(* Logix 5000 project; controller Proyecto_APM vendor 1 type 14 code 156 rev 30.11; software revision 30.00 *)

TASK MainTask (continuous, watchdog 500 ms) : MainProgram

MODULES
   Local : vendor 1 type 14 code 156 (Compact 0, rev 30.11)
      Dis : 1769-IQ16 (Compact 4, rev 1.1, Input RPI 20 ms)
      DOs : vendor 1 type 7 code 86 (Compact 5, rev 2.1, Output RPI 20 ms)
END_MODULES

VAR_GLOBAL   (* controller tags *)
   BIn : BOOL := 1;
   BoFc1 : BOOL;
   BoIn : BOOL;
   BoPi : BOOL;
   BTr : BOOL;
   CaIn : BOOL;
   EmFc : BOOL;
   EmPi : BOOL;
   FFc1 : BOOL;
   FFc2 : BOOL;
   FFc3 : BOOL;
   FiFcI : BOOL;
   FiFcS : BOOL;
   FiPi : BOOL;
   HPi : BOOL;
   I : BOOL;
   PaPi1 : BOOL;
   PaPi2 : BOOL;
   PaPi3 : BOOL;
   PaTrI : BOOL;
   PaTrS : BOOL;
   PIn : BOOL;
   S : BOOL;
END_VAR

PROGRAM MainProgram   (* main routine MainRoutine *)
VAR
   BoFc2 : BOOL;
   BoFc3 : BOOL;
   CFc1 : BOOL;
   CFc2 : BOOL;
   CFc3 : BOOL;
   E0 : BOOL := 1;
   E11_0 : BOOL := 1;
   E11_1 : BOOL;
   E11_2 : BOOL;
   E11_3 : BOOL;
   E12_0 : BOOL := 1;
   E12_1 : BOOL;
   E12_2 : BOOL;
   E12_3 : BOOL;
   E13_0 : BOOL := 1;
   E13_1 : BOOL;
   E13_2 : BOOL;
   E13_3 : BOOL;
   E2_0 : BOOL := 1;
   E2_1 : BOOL;
   E2_2 : BOOL;
   E2_3 : BOOL;
   E31_0 : BOOL := 1;
   E31_1 : BOOL;
   E31_2 : BOOL;
   E31_3 : BOOL;
   E32_0 : BOOL := 1;
   E32_1 : BOOL;
   E32_2 : BOOL;
   E32_3 : BOOL;
   E33_0 : BOOL := 1;
   E33_1 : BOOL;
   E33_2 : BOOL;
   E33_3 : BOOL;
   E3_0 : BOOL;
   E3_1 : BOOL;
   E3_2 : BOOL;
   E4_0 : BOOL;
   E4_1 : BOOL := 1;
   E4_2 : BOOL;
   E4_3 : BOOL;
   E4_4 : BOOL;
   EmIn : BOOL;
   EmTr : BOOL;
   iBIn : BOOL := 1;
   iBoFc1 : BOOL;
   iBoFc2 : BOOL;
   iBoFc3 : BOOL;
   iBoIn : BOOL;
   iBoPi : BOOL;
   iBTr : BOOL;
   iCaIn : BOOL;
   iCFc1 : BOOL;
   iCFc2 : BOOL;
   iCFc3 : BOOL;
   iEmFc : BOOL;
   iEmIn : BOOL;
   iEmPi : BOOL;
   iEmTr : BOOL;
   iFFc1 : BOOL;
   iFFc2 : BOOL;
   iFFc3 : BOOL;
   iFiFcI : BOOL;
   iFiFcS : BOOL;
   iFiPi : BOOL;
   iHPi : BOOL;
   iPaPi1 : BOOL;
   iPaPi2 : BOOL;
   iPaPi3 : BOOL;
   iPaTrI : BOOL;
   iPaTrS : BOOL;
   iPIn : BOOL;
   iRPi1 : BOOL;
   iRPi2 : BOOL;
   iRPi3 : BOOL;
   RPi1 : BOOL;
   RPi2 : BOOL;
   RPi3 : BOOL;
   Timer_1 : TIMER := (PRE := 200);
END_VAR

ROUTINE BandaTransportadora   (* ladder *)
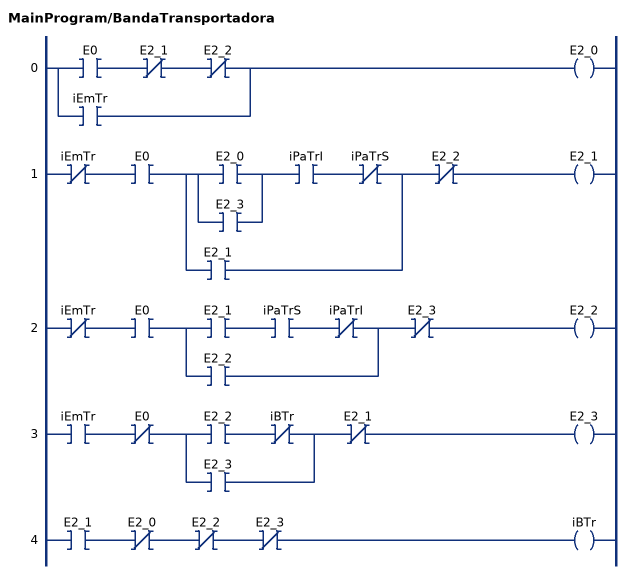
   0: [XIC(E0) XIO(E2_1) XIO(E2_2) ,XIC(iEmTr) ]OTE(E2_0);
   1: XIO(iEmTr)XIC(E0)[[XIC(E2_0) ,XIC(E2_3) ] XIC(iPaTrI) XIO(iPaTrS) ,XIC(E2_1) ]XIO(E2_2)OTE(E2_1);
   2: XIO(iEmTr)XIC(E0)[XIC(E2_1) XIC(iPaTrS) XIO(iPaTrI) ,XIC(E2_2) ]XIO(E2_3)OTE(E2_2);
   3: XIC(iEmTr)XIO(E0)[XIC(E2_2) XIO(iBTr) ,XIC(E2_3) ]XIO(E2_1)OTE(E2_3);
   4: XIC(E2_1)XIO(E2_0)XIO(E2_2)XIO(E2_3)OTE(iBTr);
END_ROUTINE

ROUTINE FresadoCortado1   (* ladder *)
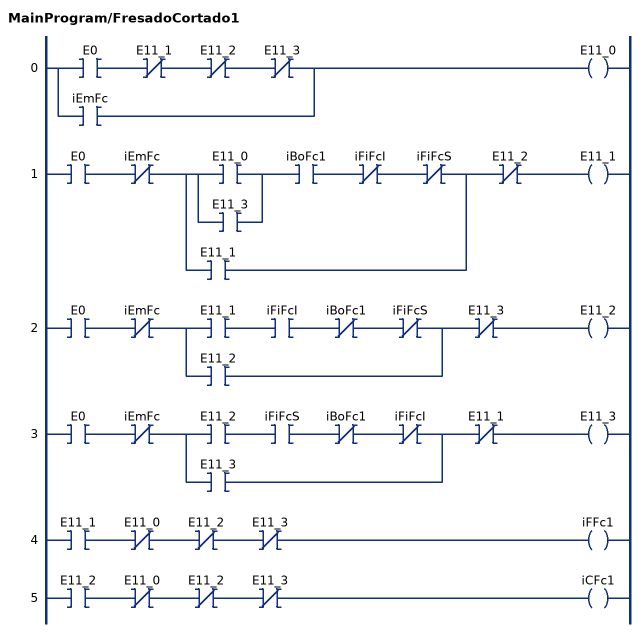
   0: [XIC(E0) XIO(E11_1) XIO(E11_2) XIO(E11_3) ,XIC(iEmFc) ]OTE(E11_0);
   1: XIC(E0)XIO(iEmFc)[[XIC(E11_0) ,XIC(E11_3) ] XIC(iBoFc1) XIO(iFiFcI) XIO(iFiFcS) ,XIC(E11_1) ]XIO(E11_2)OTE(E11_1);
   2: XIC(E0)XIO(iEmFc)[XIC(E11_1) XIC(iFiFcI) XIO(iBoFc1) XIO(iFiFcS) ,XIC(E11_2) ]XIO(E11_3)OTE(E11_2);
   3: XIC(E0)XIO(iEmFc)[XIC(E11_2) XIC(iFiFcS) XIO(iBoFc1) XIO(iFiFcI) ,XIC(E11_3) ]XIO(E11_1)OTE(E11_3);
   4: XIC(E11_1)XIO(E11_0)XIO(E11_2)XIO(E11_3)OTE(iFFc1);
   5: XIC(E11_2)XIO(E11_0)XIO(E11_2)XIO(E11_3)OTE(iCFc1);
END_ROUTINE

ROUTINE FresadoCortado2   (* ladder *)
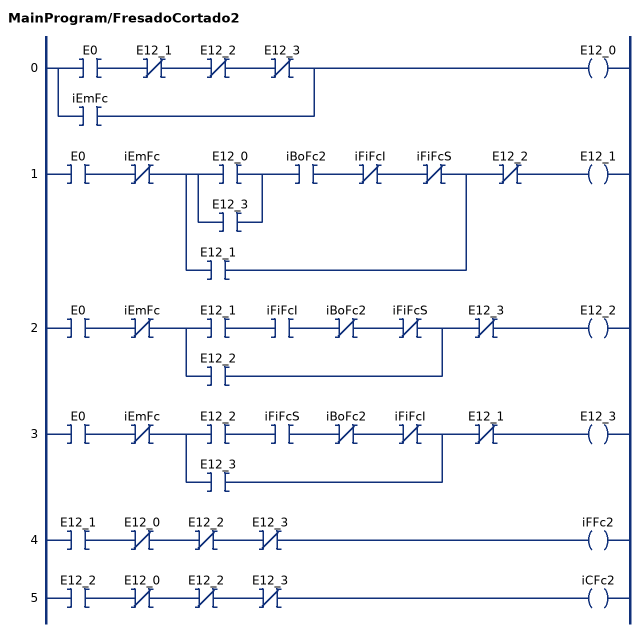
   0: [XIC(E0) XIO(E12_1) XIO(E12_2) XIO(E12_3) ,XIC(iEmFc) ]OTE(E12_0);
   1: XIC(E0)XIO(iEmFc)[[XIC(E12_0) ,XIC(E12_3) ] XIC(iBoFc2) XIO(iFiFcI) XIO(iFiFcS) ,XIC(E12_1) ]XIO(E12_2)OTE(E12_1);
   2: XIC(E0)XIO(iEmFc)[XIC(E12_1) XIC(iFiFcI) XIO(iBoFc2) XIO(iFiFcS) ,XIC(E12_2) ]XIO(E12_3)OTE(E12_2);
   3: XIC(E0)XIO(iEmFc)[XIC(E12_2) XIC(iFiFcS) XIO(iBoFc2) XIO(iFiFcI) ,XIC(E12_3) ]XIO(E12_1)OTE(E12_3);
   4: XIC(E12_1)XIO(E12_0)XIO(E12_2)XIO(E12_3)OTE(iFFc2);
   5: XIC(E12_2)XIO(E12_0)XIO(E12_2)XIO(E12_3)OTE(iCFc2);
END_ROUTINE

ROUTINE FresadoCortado3   (* ladder *)
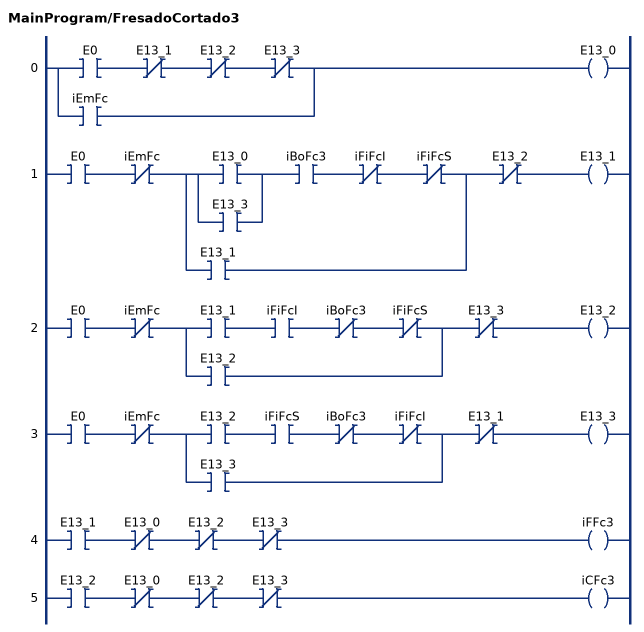
   0: [XIC(E0) XIO(E13_1) XIO(E13_2) XIO(E13_3) ,XIC(iEmFc) ]OTE(E13_0);
   1: XIC(E0)XIO(iEmFc)[[XIC(E13_0) ,XIC(E13_3) ] XIC(iBoFc3) XIO(iFiFcI) XIO(iFiFcS) ,XIC(E13_1) ]XIO(E13_2)OTE(E13_1);
   2: XIC(E0)XIO(iEmFc)[XIC(E13_1) XIC(iFiFcI) XIO(iBoFc3) XIO(iFiFcS) ,XIC(E13_2) ]XIO(E13_3)OTE(E13_2);
   3: XIC(E0)XIO(iEmFc)[XIC(E13_2) XIC(iFiFcS) XIO(iBoFc3) XIO(iFiFcI) ,XIC(E13_3) ]XIO(E13_1)OTE(E13_3);
   4: XIC(E13_1)XIO(E13_0)XIO(E13_2)XIO(E13_3)OTE(iFFc3);
   5: XIC(E13_2)XIO(E13_0)XIO(E13_2)XIO(E13_3)OTE(iCFc3);
END_ROUTINE

ROUTINE Inspeccin   (* ladder *)
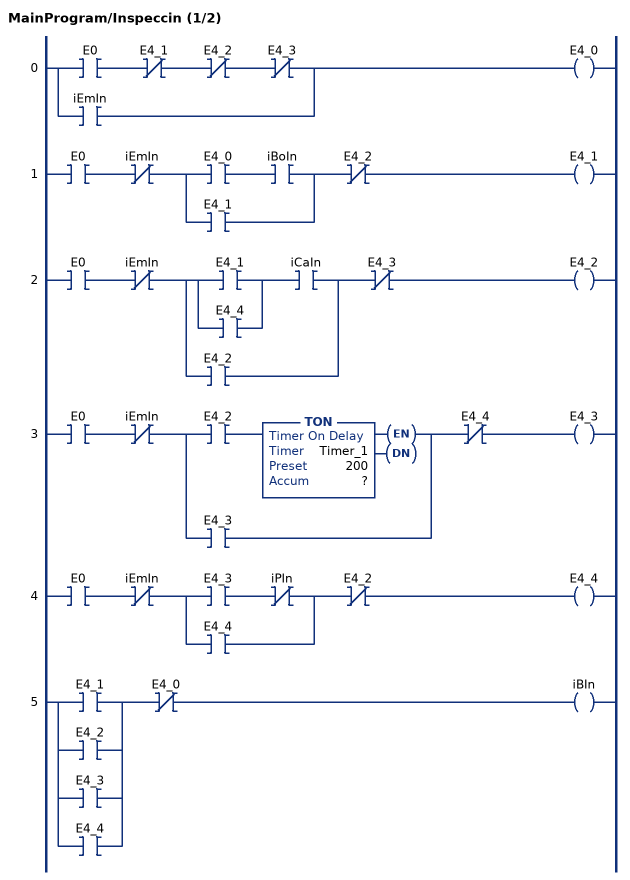
   0: [XIC(E0) XIO(E4_1) XIO(E4_2) XIO(E4_3) ,XIC(iEmIn) ]OTE(E4_0);
   1: XIC(E0)XIO(iEmIn)[XIC(E4_0) XIC(iBoIn) ,XIC(E4_1) ]XIO(E4_2)OTE(E4_1);
   2: XIC(E0)XIO(iEmIn)[[XIC(E4_1) ,XIC(E4_4) ] XIC(iCaIn) ,XIC(E4_2) ]XIO(E4_3)OTE(E4_2);
   3: XIC(E0)XIO(iEmIn)[XIC(E4_2) TON(Timer_1,?,?) ,XIC(E4_3) ]XIO(E4_4)OTE(E4_3);
   4: XIC(E0)XIO(iEmIn)[XIC(E4_3) XIO(iPIn) ,XIC(E4_4) ]XIO(E4_2)OTE(E4_4);
   5: [XIC(E4_1) ,XIC(E4_2) ,XIC(E4_3) ,XIC(E4_4) ]XIO(E4_0)OTE(iBIn);
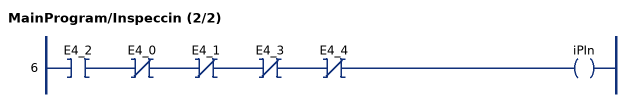
   6: XIC(E4_2)XIO(E4_0)XIO(E4_1)XIO(E4_3)XIO(E4_4)OTE(iPIn);
END_ROUTINE

ROUTINE MainRoutine   (* ladder *)
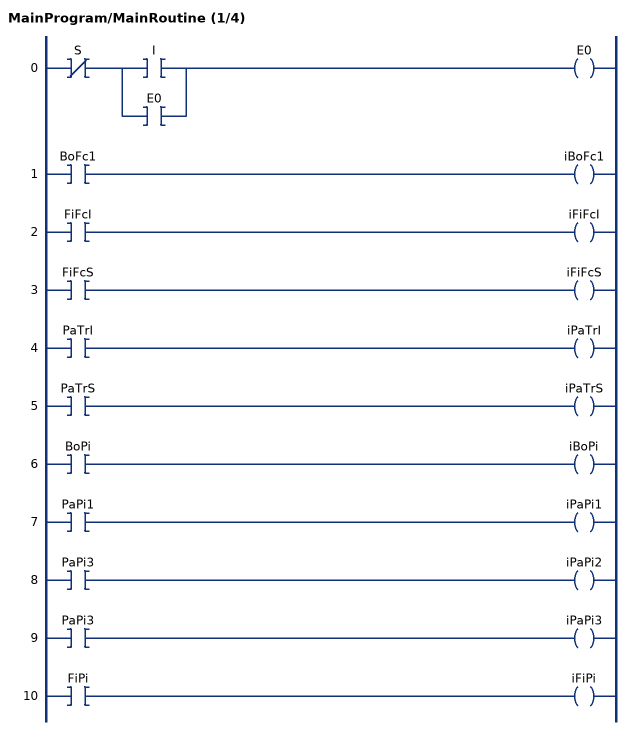
   0: XIO(S)[XIC(I) ,XIC(E0) ]OTE(E0);
   1: XIC(BoFc1)OTE(iBoFc1);
   2: XIC(FiFcI)OTE(iFiFcI);
   3: XIC(FiFcS)OTE(iFiFcS);
   4: XIC(PaTrI)OTE(iPaTrI);
   5: XIC(PaTrS)OTE(iPaTrS);
   6: XIC(BoPi)OTE(iBoPi);
   7: XIC(PaPi1)OTE(iPaPi1);
   8: XIC(PaPi3)OTE(iPaPi2);
   9: XIC(PaPi3)OTE(iPaPi3);
   10: XIC(FiPi)OTE(iFiPi);
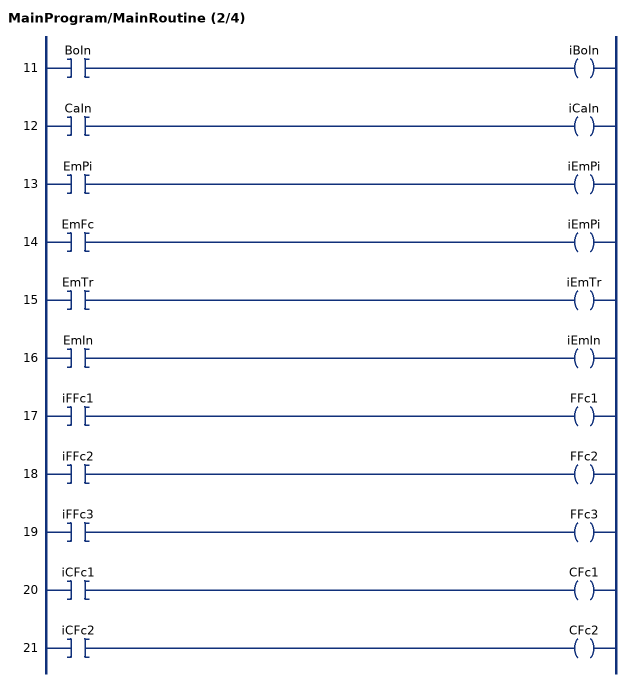
   11: XIC(BoIn)OTE(iBoIn);
   12: XIC(CaIn)OTE(iCaIn);
   13: XIC(EmPi)OTE(iEmPi);
   14: XIC(EmFc)OTE(iEmPi);
   15: XIC(EmTr)OTE(iEmTr);
   16: XIC(EmIn)OTE(iEmIn);
   17: XIC(iFFc1)OTE(FFc1);
   18: XIC(iFFc2)OTE(FFc2);
   19: XIC(iFFc3)OTE(FFc3);
   20: XIC(iCFc1)OTE(CFc1);
   21: XIC(iCFc2)OTE(CFc2);
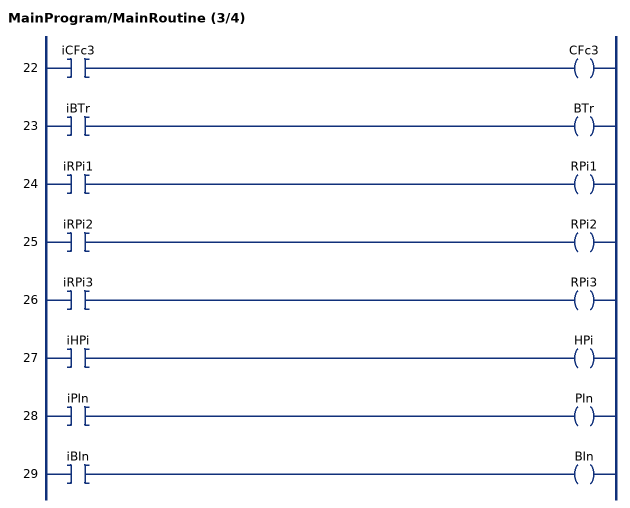
   22: XIC(iCFc3)OTE(CFc3);
   23: XIC(iBTr)OTE(BTr);
   24: XIC(iRPi1)OTE(RPi1);
   25: XIC(iRPi2)OTE(RPi2);
   26: XIC(iRPi3)OTE(RPi3);
   27: XIC(iHPi)OTE(HPi);
   28: XIC(iPIn)OTE(PIn);
   29: XIC(iBIn)OTE(BIn);
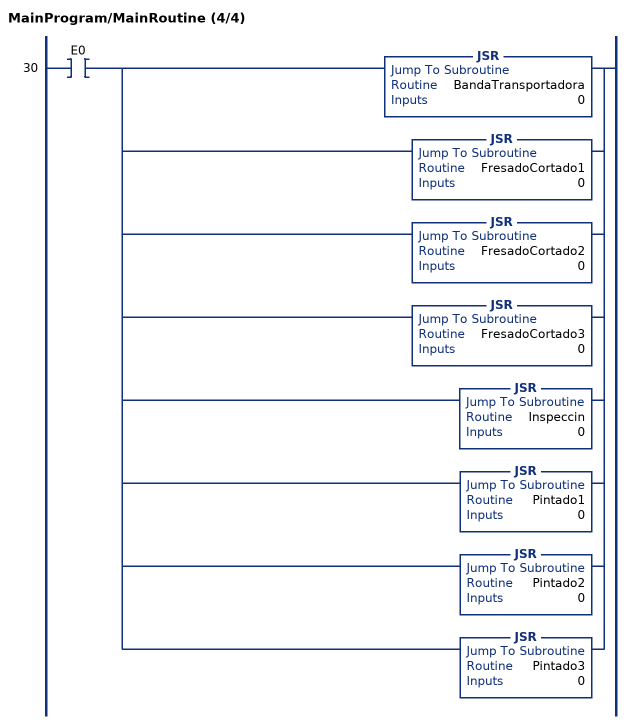
   30: XIC(E0)[JSR(BandaTransportadora,0) ,JSR(FresadoCortado1,0) ,JSR(FresadoCortado2,0) ,JSR(FresadoCortado3,0) ,JSR(Inspeccin,0) ,JSR(Pintado1,0) ,JSR(Pintado2,0) ,JSR(Pintado3,0) ];
END_ROUTINE

ROUTINE Pintado1   (* ladder *)
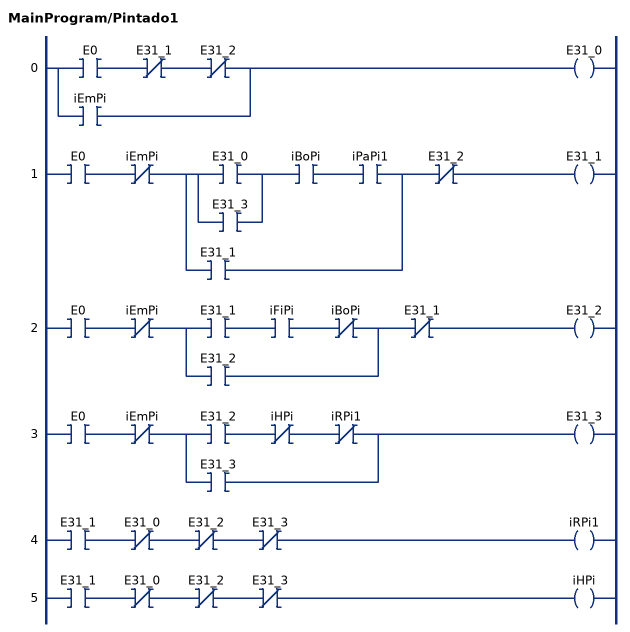
   0: [XIC(E0) XIO(E31_1) XIO(E31_2) ,XIC(iEmPi) ]OTE(E31_0);
   1: XIC(E0)XIO(iEmPi)[[XIC(E31_0) ,XIC(E31_3) ] XIC(iBoPi) XIC(iPaPi1) ,XIC(E31_1) ]XIO(E31_2)OTE(E31_1);
   2: XIC(E0)XIO(iEmPi)[XIC(E31_1) XIC(iFiPi) XIO(iBoPi) ,XIC(E31_2) ]XIO(E31_1)OTE(E31_2);
   3: XIC(E0)XIO(iEmPi)[XIC(E31_2) XIO(iHPi) XIO(iRPi1) ,XIC(E31_3) ]OTE(E31_3);
   4: XIC(E31_1)XIO(E31_0)XIO(E31_2)XIO(E31_3)OTE(iRPi1);
   5: XIC(E31_1)XIO(E31_0)XIO(E31_2)XIO(E31_3)OTE(iHPi);
END_ROUTINE

ROUTINE Pintado2   (* ladder *)
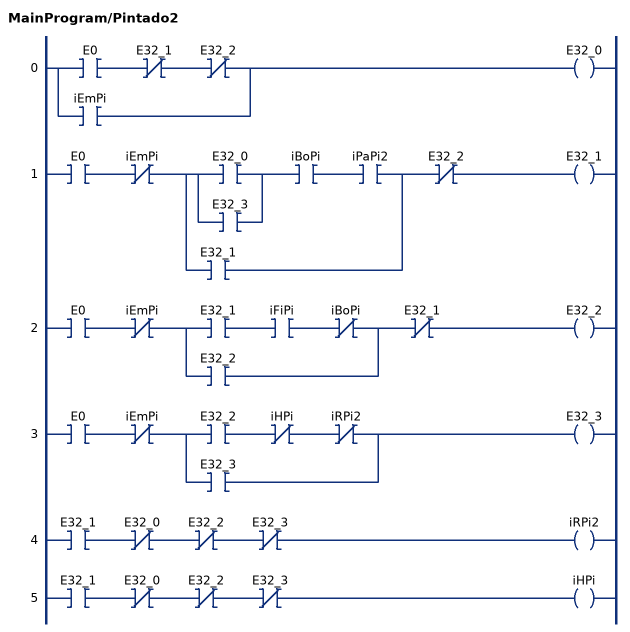
   0: [XIC(E0) XIO(E32_1) XIO(E32_2) ,XIC(iEmPi) ]OTE(E32_0);
   1: XIC(E0)XIO(iEmPi)[[XIC(E32_0) ,XIC(E32_3) ] XIC(iBoPi) XIC(iPaPi2) ,XIC(E32_1) ]XIO(E32_2)OTE(E32_1);
   2: XIC(E0)XIO(iEmPi)[XIC(E32_1) XIC(iFiPi) XIO(iBoPi) ,XIC(E32_2) ]XIO(E32_1)OTE(E32_2);
   3: XIC(E0)XIO(iEmPi)[XIC(E32_2) XIO(iHPi) XIO(iRPi2) ,XIC(E32_3) ]OTE(E32_3);
   4: XIC(E32_1)XIO(E32_0)XIO(E32_2)XIO(E32_3)OTE(iRPi2);
   5: XIC(E32_1)XIO(E32_0)XIO(E32_2)XIO(E32_3)OTE(iHPi);
END_ROUTINE

ROUTINE Pintado3   (* ladder *)
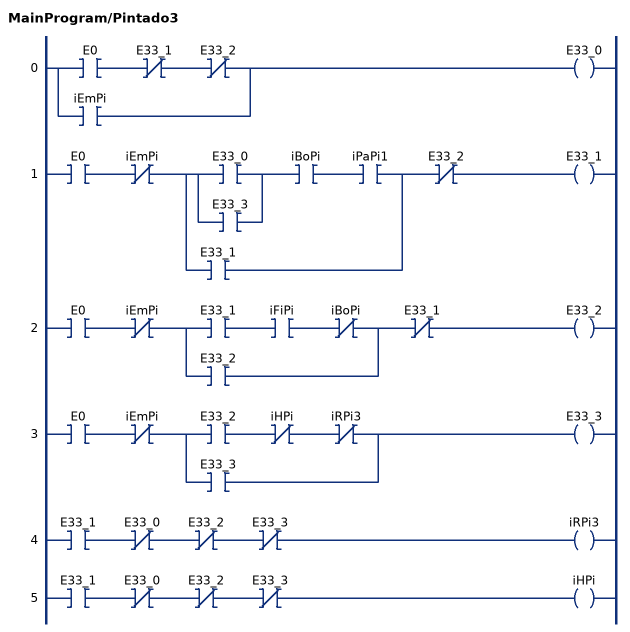
   0: [XIC(E0) XIO(E33_1) XIO(E33_2) ,XIC(iEmPi) ]OTE(E33_0);
   1: XIC(E0)XIO(iEmPi)[[XIC(E33_0) ,XIC(E33_3) ] XIC(iBoPi) XIC(iPaPi1) ,XIC(E33_1) ]XIO(E33_2)OTE(E33_1);
   2: XIC(E0)XIO(iEmPi)[XIC(E33_1) XIC(iFiPi) XIO(iBoPi) ,XIC(E33_2) ]XIO(E33_1)OTE(E33_2);
   3: XIC(E0)XIO(iEmPi)[XIC(E33_2) XIO(iHPi) XIO(iRPi3) ,XIC(E33_3) ]OTE(E33_3);
   4: XIC(E33_1)XIO(E33_0)XIO(E33_2)XIO(E33_3)OTE(iRPi3);
   5: XIC(E33_1)XIO(E33_0)XIO(E33_2)XIO(E33_3)OTE(iHPi);
END_ROUTINE
END_PROGRAM
